FUNCTION_BLOCK Real5_Array (* Basic FB with empty ECC *)
  (* Standard: 61499-2 *)
  (* Version 1.0, 2020-08-13, Candra Wardaya, UGM *)
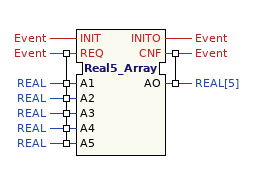
  EVENT_INPUT
    INIT; (* Initial Trigger *)
    REQ WITH A1, A2, A3, A4, A5; (* Execution Request *)
  END_EVENT
  EVENT_OUTPUT
    INITO; (* Output Initialization *)
    CNF WITH AO; (* Confirmation of Execution *)
  END_EVENT
  VAR_INPUT
    A1 : REAL; (* Single Real Input *)
    A2 : REAL; (* Single Real Input *)
    A3 : REAL; (* Single Real Input *)
    A4 : REAL; (* Single Real Input *)
    A5 : REAL; (* Single Real Input *)
  END_VAR
  VAR_OUTPUT
    AO : ARRAY [0..4] OF REAL; (* Array Output *)
  END_VAR
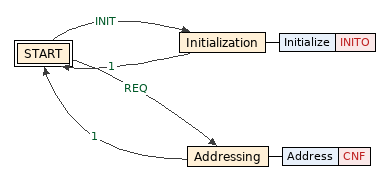
  EC_STATES
    START; (* Initial State *)
    Initialization : Initialize -> INITO;
    Addressing : Address -> CNF;
  END_STATES
  EC_TRANSITIONS
    START TO Initialization := INIT;
    Initialization TO START := 1;
    START TO Addressing := REQ;
    Addressing TO START := 1;
  END_TRANSITIONS
  ALGORITHM Initialize IN ST: (* New Algorithm *)

  END_ALGORITHM
  ALGORITHM Address IN ST: (* New Algorithm *)
AO[0] := A1;
AO[1] := A2;
AO[2] := A3;
AO[3] := A4;
AO[4] := A5;
  END_ALGORITHM
END_FUNCTION_BLOCK
